// TIA Portal V19 export
TYPE "LEXCHANGETRAY_typeHandlingXyzEm_deliver_interface"
// stored: Access Published
   STRUCT
      init : Bool;
      constraintRoller : "LEXCHANGETRAY_typeHandlingXyzEm_toConstraintRollerDeliver";
      plasticRoller { S7_SetPoint := 'True'} : "LEXCHANGETRAY_typeHandlingXyzEm_toPlasticDeliver";
      NgConvyorRoller { S7_SetPoint := 'True'} : "LEXCHANGETRAY_typeHandlingXyzEm_toNgConveyorDeliver";
   END_STRUCT;
END_TYPE
